SYSTEM openCVtest
  (* Version 1.0, 2026-06-16, alex *)
  APPLICATION openCVtestApp
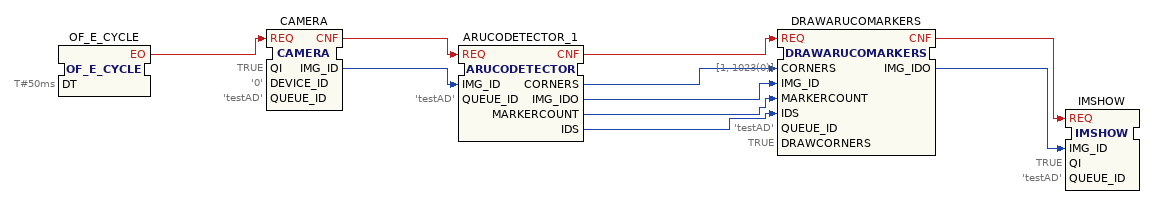
    FBS
      IMSHOW : IMSHOW(QI := TRUE, QUEUE_ID := 'testAD');
      DRAWARUCOMARKERS : DRAWARUCOMARKERS(QUEUE_ID := 'testAD', CORNERS := [1, 1023(0)], DRAWCORNERS := TRUE);
      ARUCODETECTOR_1 : ARUCODETECTOR(QUEUE_ID := 'testAD');
      CAMERA : CAMERA(QI := TRUE, DEVICE_ID := '0', QUEUE_ID := 'testAD');
      OF_E_CYCLE : OF_E_CYCLE(DT := T#50ms);
    END_FBS
    EVENT_CONNECTIONS
      DRAWARUCOMARKERS.CNF TO IMSHOW.REQ;
      ARUCODETECTOR_1.CNF TO DRAWARUCOMARKERS.REQ;
      CAMERA.CNF TO ARUCODETECTOR_1.REQ;
      OF_E_CYCLE.EO TO CAMERA.REQ;
    END_CONNECTIONS
    DATA_CONNECTIONS
      DRAWARUCOMARKERS.IMG_IDO TO IMSHOW.IMG_ID;
      ARUCODETECTOR_1.CORNERS TO DRAWARUCOMARKERS.CORNERS;
      ARUCODETECTOR_1.IMG_IDO TO DRAWARUCOMARKERS.IMG_ID;
      CAMERA.IMG_ID TO ARUCODETECTOR_1.IMG_ID;
      ARUCODETECTOR_1.MARKERCOUNT TO DRAWARUCOMARKERS.MARKERCOUNT;
      ARUCODETECTOR_1.IDS TO DRAWARUCOMARKERS.IDS;
    END_CONNECTIONS
  END_APPLICATION
  DEVICE FORTE_PC : FORTE_PC(MGR_ID := "localhost:61499" (* Device manager socket ID *))
    {SET_ATTRIBUTE(Profile, HOLOBLOC)}
    RESOURCE EMB_RES : EMB_RES
    END_RESOURCE
  END_DEVICE
  MAPPINGS
    openCVtestApp.IMSHOW ON FORTE_PC.EMB_RES;
    openCVtestApp.DRAWARUCOMARKERS ON FORTE_PC.EMB_RES;
    openCVtestApp.ARUCODETECTOR_1 ON FORTE_PC.EMB_RES;
    openCVtestApp.CAMERA ON FORTE_PC.EMB_RES;
    openCVtestApp.OF_E_CYCLE ON FORTE_PC.EMB_RES;
  END_MAPPINGS
  SEGMENTS
    Ethernet : Ethernet;
  END_SEGMENTS
  LINKS
    FORTE_PC => Ethernet;
  END_LINKS
END_SYSTEM
